// TIA Portal V20 export
// export: Created 2026-10-03T18:54:34.6248224Z, ExportSetting WithDefaults, DisplayName Totally Integrated Automation Portal, DisplayVersion V20 Update 4, DisplayName TIA Portal Openness, DisplayVersion V20 Update 4, DisplayName TIA Portal Version Control Interface, DisplayVersion V20 Update 4, DisplayName SINAMICS Startdrive Advanced, DisplayVersion V20 SP1 Update 1, DisplayName SINAMICS Startdrive G110M, G120, G120C, G120D, G120P, G115D, DisplayVersion V20 SP1 Update 1, DisplayName SINAMICS Startdrive G130, G150, S120, S150, SINAMICS MV, G220, S200, S210, DisplayVersion V20 SP1 Update 1, DisplayName STEP 7 Professional, DisplayVersion V20 Update 4, DisplayName STEP 7 Safety, DisplayVersion V20 Update 2, DisplayName WinCC Basic/Comfort/Advanced, DisplayVersion V20 Update 4, DisplayName WinCC Unified, DisplayVersion V20 Update 4
FUNCTION "SLC_BIT_RESET" : Void   // FC20, SCL
TITLE = Reset (unlatch) a bit by file, element and bit number
{ S7_Optimized_Access := 'TRUE' }
VERSION : 0.1
// Replaces OTU on an indirect bit address such as B3:70/[N7:200].
// stored: AutoNumber true, IsIECCheckEnabled false, SetENOAutomatically false, UDAEnableTagReadback false
   VAR_INPUT
      File : DInt;   // Data file number (3 for B3)
      Element : DInt;   // Word number
      Bit : DInt;   // Bit number
   END_VAR
BEGIN
   // Words are stored high byte first, so bits 8-15 are in the first byte and bits 0-7 in the second.
   POKE_BOOL(area := 16#84, dbNumber := #File,
             byteOffset := (#Element + #Bit / 16) * 2 + SEL(G := (#Bit MOD 16) >= 8, IN0 := 1, IN1 := 0),
             bitOffset := #Bit MOD 8, value := FALSE);
END_FUNCTION
